{attribute 'GeneratedUsingTerminal: EL2912-0000-0016'}
{attribute addProperty BoxType "EL2912-0000-0016"}
{attribute addProperty Id "FSOEAT %Q*FSOE_F76352459"}
{attribute addProperty CRC "949596549"}
{attribute addProperty Size "9"}
TYPE FSoE_Outputs_3899B185 :
STRUCT
	{attribute addProperty Name "FSOE"}
	FSOE AT %Q* : FSOE_F7635245;
END_STRUCT
END_TYPE

(* stored: Version 1.2.0.0, ProductVersion 3.1.4024.9
   DUT FSoE_Outputs_3899B185: Id {2e13d7df-6ffc-4bbd-b617-575193bc3915} *)
